PROGRAM MAIN
VAR
END_VAR

END_PROGRAM

(* stored: Version 1.1.0.1
   POU MAIN: Id {34cfb158-ade0-4c46-a4eb-2ee3bc202923} *)
